VAR_GLOBAL
	packTags	:	ST_PackMLv30;
END_VAR

(* stored: Version 1.1.0.1, ProductVersion 3.1.4022.16
   GVL GV: Id {16eb9ac4-571c-49b1-a239-4495c5201a54} *)
